TYPE
   ST_SymbolHandle :
   STRUCT
      Handle : DWORD;
      SymbolAddress : ST_SymbolAddress;
   END_STRUCT
END_TYPE

(* stored: Version 1.1.0.1, ProductVersion 3.1.4024.9
   DUT ST_SymbolHandle: Id {6b63cd5d-7aae-448d-a69a-edd770a10da9} *)
